Staubli VAL3: AA_Chessie.dtx

jointRx jStart = {j1=-4.35, j2=22.39, j3=131, j5=25.77, j6=50.65}
jointRx jDepart = {j1=20.811233, j2=126.617326, j3=-10.855704, j5=64.238378, j6=-69.188767}
frame fFrame = {x=374.8, y=3.07, z=-517.036829, rx=-180, fatherId=world[0]}
pointRx pTable = {fatherId=fFrame[0]}
pointRx pCaseNoire[33]
  [0] = {x=374.8, y=3.07, z=-517.036829, rx=-180, shoulder=lefty, elbow=epositive, wrist=wpositive, fatherId=world[0]}
  [1] = {fatherId=world[0]}
  [2] = {fatherId=world[0]}
  [3] = {fatherId=world[0]}
  [4] = {fatherId=world[0]}
  [5] = {fatherId=world[0]}
  [6] = {fatherId=world[0]}
  [7] = {fatherId=world[0]}
  [8] = {fatherId=world[0]}
  [9] = {fatherId=world[0]}
  [10] = {fatherId=world[0]}
  [11] = {fatherId=world[0]}
  [12] = {fatherId=world[0]}
  [13] = {fatherId=world[0]}
  [14] = {fatherId=world[0]}
  [15] = {fatherId=world[0]}
  [16] = {fatherId=world[0]}
  [17] = {fatherId=world[0]}
  [18] = {fatherId=world[0]}
  [19] = {fatherId=world[0]}
  [20] = {fatherId=world[0]}
  [21] = {fatherId=world[0]}
  [22] = {fatherId=world[0]}
  [23] = {fatherId=world[0]}
  [24] = {fatherId=world[0]}
  [25] = {fatherId=world[0]}
  [26] = {fatherId=world[0]}
  [27] = {fatherId=world[0]}
  [28] = {fatherId=world[0]}
  [29] = {fatherId=world[0]}
  [30] = {fatherId=world[0]}
  [31] = {fatherId=world[0]}
  [32] = {fatherId=world[0]}
jointRx jCaseNoire = {j1=-7.236149, j2=83.896154, j3=110.243942, j5=-14.140096, j6=172.763851}
num nX
num nY
num ni
mdesc mPrise = {accel=25}
mdesc mDepose = {accel=25}
mdesc mDeplacement = {accel=250}
tool tTool = {x=2.67332365613152, y=0.0823457375943404, z=50.1043771229301, rx=-7.34240987449236E-12, ry=-8.49495425328202E-12, rz=2.13111140704977E-13, fatherId=flange[0], ioLink=valve1}
jointRx jInitial
trsf trAppro = {z=-10}
